// TIA Portal project "FactoryIO_scene3" (V16)

(* hardware
DEVICE "S7-1200 station_1"  S7-1200 Station
   slot 0: "Rack_0"  S7-1200 Rack  Rack  V1.0
   slot 1: "PLC_1"  CPU 1214C DC/DC/DC  6ES7 214-1AG40-0XB0  V4.4
*)

// ===== PLC "PLC_1"  CPU 1214C DC/DC/DC =====

VAR_GLOBAL   // PLC tag table "Default tag table"
   "Tag_1" AT %M0.0 : Bool;
   "Tag_2" AT %M0.1 : Bool;
   "Tag_3" AT %M0.2 : Bool;
END_VAR

VAR_GLOBAL   // PLC tag table "IO_tags"
   "Item ready" AT %I0.0 : Bool;
   "At Entry" AT %I0.1 : Bool;
   "At Exit" AT %I0.2 : Bool;
   "Factory IO running" AT %I0.3 : Bool;
   "Entry Conveyor" AT %Q0.0 : Bool;
   "Buffer Conveyor" AT %Q0.1 : Bool;
   "Emitter" AT %Q0.2 : Bool;
   "Remover" AT %Q0.3 : Bool;
END_VAR

DATA_BLOCK "data"   // DB4
{ S7_Optimized_Access := 'TRUE' }
VERSION : 0.1
   VAR
      reset : Bool;
   END_VAR
BEGIN
END_DATA_BLOCK

// folder: System blocks/Program resources

DATA_BLOCK "Entry_Counter_0_DB"   // DB1
{ S7_Optimized_Access := 'TRUE' }
AUTHOR : Simatic
FAMILY : IEC
NAME : CNTR
VERSION : 1.0
// stored: InstanceOfName IEC_COUNTER
"IEC_COUNTER"
BEGIN
END_DATA_BLOCK

DATA_BLOCK "Item_Counter_0_DB"   // DB2
{ S7_Optimized_Access := 'TRUE' }
AUTHOR : Simatic
FAMILY : IEC
NAME : CNTR
VERSION : 1.0
// stored: InstanceOfName IEC_COUNTER
"IEC_COUNTER"
BEGIN
END_DATA_BLOCK

DATA_BLOCK "Exit_Counter_0_DB"   // DB3
{ S7_Optimized_Access := 'TRUE' }
AUTHOR : Simatic
FAMILY : IEC
NAME : CNTR
VERSION : 1.0
// stored: InstanceOfName IEC_COUNTER
"IEC_COUNTER"
BEGIN
END_DATA_BLOCK

// folder: (top level)

FUNCTION "MHJ-PLC-Lab-Function-S71200" : Void   // FC9000, SCL
{ S7_Optimized_Access := 'TRUE' }
VERSION : 0.1
   VAR_TEMP
      rdTimeReturn : Int;
      outputTime : DTL;
      SyncVal : Byte;
      forVal : Int;
      forVal_2 : Int;
      Value : Byte;
   END_VAR
   VAR CONSTANT
      CompVal : Byte := 16#34;
      Value_01 : Byte := 16#11;
      Value_01_DW : DWord := 16#A165_D992;
      Value_02_DW : DWord := 16#58BE_4401;
   END_VAR
BEGIN

   #Value:=PEEK(area := 16#82,
        dbNumber := 0,
        byteOffset := 511);
   #Value := #Value + 1;

   POKE(area := 16#82,
        dbNumber := 0,
        byteOffset := 511,
        value := #Value);

   POKE(area:=16#81,
        dbNumber:=0,
        byteOffset:=1016,
        value:=#Value_01_DW);
   POKE(area := 16#81,
        dbNumber := 0,
        byteOffset := 1020,
        value := #Value_02_DW);

   POKE(area := 16#81,
        dbNumber := 0,
        byteOffset := 511,
        value := B#16#00);

   FOR #forVal := 0 TO 120 DO
       FOR #forVal_2:=0 TO 10 DO
           #rdTimeReturn:=RD_SYS_T(#outputTime);
           #rdTimeReturn := WR_SYS_T(#outputTime);
           #rdTimeReturn := RD_SYS_T(#outputTime);
           #rdTimeReturn := WR_SYS_T(#outputTime);
       END_FOR;
       #SyncVal:= PEEK(area := 16#81,
                      dbNumber := 0,
                      byteOffset := 511);
       IF #SyncVal = #CompVal THEN
          GOTO M_1;
       END_IF;
   END_FOR;
   RETURN;

   M_1:
   POKE(area := 16#81,
        dbNumber := 0,
        byteOffset := 511,
        value := B#16#0);
END_FUNCTION

ORGANIZATION_BLOCK "Main"   // OB1, LAD, ProgramCycle
TITLE = "Main Program Sweep (Cycle)"
{ S7_Optimized_Access := 'TRUE' }
VERSION : 0.1
   VAR_INPUT
      Initial_Call : Bool;   // Initial call of this OB
      Remanence : Bool;   // =True, if remanent data are available
   END_VAR
   VAR_TEMP
      current_step : Int;
      reset : Bool;
   END_VAR
   VAR CONSTANT
      box_count : Int := 3;   // Number of buffer boxes
   END_VAR
   VAR_TEMP   // added for the SCL form of the ladder/FBD networks
      _w1 : Bool;
   END_VAR
BEGIN

REGION Network 1
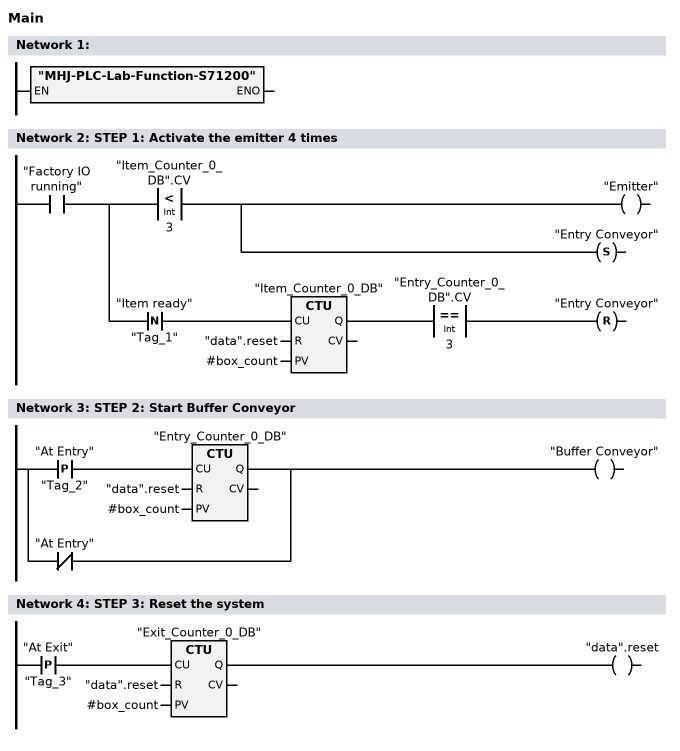
   RUNG wire#powerrail
      "MHJ-PLC-Lab-Function-S71200"()
   END_RUNG
   // the same network as SCL:
   "MHJ-PLC-Lab-Function-S71200"();
END_REGION

REGION Network 2: STEP 1: Activate the emitter 4 times
   "Emitter" := "Factory IO running" AND ("Item_Counter_0_DB".CV < 3);
   IF "Emitter" THEN "Entry Conveyor" := TRUE; END_IF;
   #_w1 := "Factory IO running" AND NOT "Item ready" AND "Tag_1";   // falling edge of "Item ready"
   "Tag_1" := "Item ready";
   "Item_Counter_0_DB".CTU(CU := #_w1, R := "data".reset, PV := #box_count);
   IF "Item_Counter_0_DB".Q AND ("Entry_Counter_0_DB".CV = 3) THEN "Entry Conveyor" := FALSE; END_IF;
END_REGION

REGION Network 3: STEP 2: Start Buffer Conveyor
   #_w1 := "At Entry" AND NOT "Tag_2";   // rising edge of "At Entry"
   "Tag_2" := "At Entry";
   "Entry_Counter_0_DB".CTU(CU := #_w1, R := "data".reset, PV := #box_count);
   "Buffer Conveyor" := "Entry_Counter_0_DB".Q OR NOT "At Entry";
END_REGION

REGION Network 4: STEP 3: Reset the system
   #_w1 := "At Exit" AND NOT "Tag_3";   // rising edge of "At Exit"
   "Tag_3" := "At Exit";
   "Exit_Counter_0_DB".CTU(CU := #_w1, R := "data".reset, PV := #box_count);
   "data".reset := "Exit_Counter_0_DB".Q;
END_REGION
END_ORGANIZATION_BLOCK